PROGRAM MAIN
VAR
END_VAR

END_PROGRAM

(* stored: Version 1.1.0.1, ProductVersion 3.1.4024.12
   POU MAIN: Id {90b89767-3bdb-45b8-891a-e1dd770f9097}, SpecialFunc None *)
